(* Logix 5000 project; controller APM20233008 vendor 1 type 14 code 156 rev 30.11; software revision 30.00 *)

TASK MainTask (continuous, watchdog 500 ms) : MainProgram

MODULES
   Local : vendor 1 type 14 code 156 (Compact 0, rev 30.11)
      DIN : 1769-IQ16 (Compact 4, rev 1.1, Input RPI 20 ms)
      DOUT : vendor 1 type 7 code 86 (Compact 5, rev 2.1, Output RPI 20 ms)
END_MODULES

VAR_GLOBAL   (* controller tags *)
   ALARMA : BOOL;
   BANDA : ALIAS FOR Local:5:O.Data.0;
   LOTEOK : BOOL;
   PIEZASP : COUNTER := (PRE := 8);
   RESET_LOTE : BOOL;
   ROBOT : BOOL;
   SCADA_START_BANDA : BOOL;
   SCADA_STOP_BANDA : BOOL;
   SENSOR_PIEZA : BOOL;
   START_BANDA : ALIAS FOR Local:4:I.Data.1;
   START_RUTINA_ROBOT : BOOL;
   STOP_BANDA : ALIAS FOR Local:4:I.Data.0;
   STOP_RUTINA_ROBOT : BOOL;
END_VAR

PROGRAM MainProgram   (* main routine MainRoutine *)

ROUTINE MainRoutine   (* ladder *)
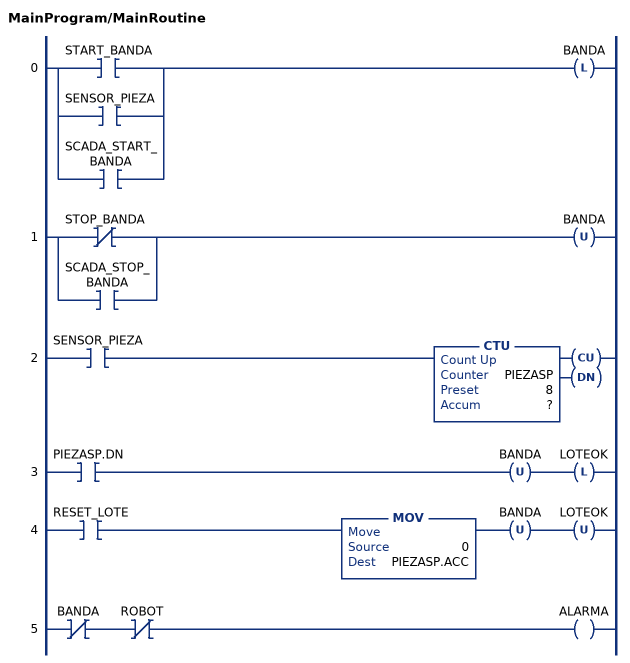
   0: [XIC(START_BANDA) ,XIC(SENSOR_PIEZA) ,XIC(SCADA_START_BANDA) ]OTL(BANDA);
   1: [XIO(STOP_BANDA) ,XIC(SCADA_STOP_BANDA) ]OTU(BANDA);
   2: XIC(SENSOR_PIEZA)CTU(PIEZASP,?,?);
   3: XIC(PIEZASP.DN)OTU(BANDA)OTL(LOTEOK);
   4: XIC(RESET_LOTE)MOV(0,PIEZASP.ACC)OTU(BANDA)OTU(LOTEOK);
   5: XIO(BANDA)XIO(ROBOT)OTE(ALARMA);
END_ROUTINE
END_PROGRAM
